FUNCTION_BLOCK PAMSilo EXTENDS PAProcessModule IMPLEMENTS IPAMSilo
VAR_INPUT
END_VAR
VAR_OUTPUT
END_VAR
VAR
	_PAPointMatIn1 : PAPoint(THIS^);
	_PAPointMatOut1 : PAPoint(THIS^);
END_VAR

METHOD FB_init : BOOL
VAR_INPUT
	bInitRetains : BOOL; // if TRUE, the retain variables are initialized (warm start / cold start)
	bInCopyCode : BOOL;  // if TRUE, the instance afterwards gets moved into the copy code (online change)
	parent : IACComponent;
END_VAR
AddPoint(_PAPointMatIn1);
AddPoint(_PAPointMatOut1);
END_METHOD

PROPERTY PUBLIC PAPointMatIn1 : IACPoint
GET
PAPointMatIn1 := _PAPointMatIn1;
END_GET
END_PROPERTY

PROPERTY PUBLIC PAPointMatOut1 : IACPoint
GET
PAPointMatOut1 := _PAPointMatOut1;
END_GET
END_PROPERTY

END_FUNCTION_BLOCK

(* stored: Version 1.1.0.1, ProductVersion 3.1.4020.12
   POU PAMSilo: Id {8c438af7-c522-409b-9349-cd0efcda1a63}, SpecialFunc None
   Method FB_init: Id {b6179cc6-bc46-48f1-9547-def2a8758866}
   Property PAPointMatIn1: Id {e98b3327-6e29-46d9-82cc-f3779057e7e3}
   Get Get: Id {39bc2f33-fa15-4235-9675-52bf2318a5b3}
   Property PAPointMatOut1: Id {92538e8c-a0aa-4e7e-9103-01f97295cbf1}
   Get Get: Id {ebcb0c74-154a-4c6c-8e90-9aa04a7d4d5b} *)
